{attribute 'linkalways'} 
{attribute 'no_explicit_call' := 'This FB is a CLASS and must be accessed using methods or properties'}
{attribute 'enable_dynamic_creation'}
FUNCTION_BLOCK _USINT EXTENDS NumericDatatypeBase
VAR
	localData : USINT;
	activeData : REFERENCE TO USINT REF= localData;
END_VAR

PROPERTY PUBLIC Address : PVOID
GET
Address := ADR(activeData);
END_GET
END_PROPERTY

METHOD PUBLIC ClearReference
VAR_INPUT
END_VAR
activeData REF= localData;
END_METHOD

METHOD PUBLIC Clone : I_Datatype
VAR
    pClone : POINTER TO _USINT;
END_VAR
pClone := __NEW(_USINT(InitialValue := Value));
Clone := pClone^;
END_METHOD

METHOD FB_init : BOOL
VAR_INPUT
	bInitRetains : BOOL; // if TRUE, the retain variables are initialized (warm start / cold start)
	bInCopyCode : BOOL;  // if TRUE, the instance afterwards gets moved into the copy code (online change)
	InitialValue : USINT;
END_VAR
localData := InitialValue;
END_METHOD

PROPERTY PUBLIC IsEven : BOOL
GET
IsEven := (Value mod 2) = 0;
END_GET
END_PROPERTY

PROPERTY PUBLIC IsFloat : BOOL
GET
IsFloat := FALSE;
END_GET
END_PROPERTY

PROPERTY PUBLIC IsSigned : BOOL
GET
IsSigned := FALSE;
END_GET
END_PROPERTY

METHOD PUBLIC MakeReferenceTo
VAR_INPUT
	ReferenceTarget : REFERENCE TO USINT;
END_VAR
activeData REF= ReferenceTarget;
END_METHOD

PROPERTY PUBLIC MaxValue : USINT
GET
MaxValue :=  DatatypeLimits.USINT_MAX_VALUE;
END_GET
END_PROPERTY

PROPERTY PUBLIC MinValue : USINT
GET
MinValue := DatatypeLimits.USINT_MIN_VALUE;
END_GET
END_PROPERTY

METHOD PROTECTED SerializeMaxValue
VAR_INPUT
	Serializer : I_Serializer;
END_VAR
Serializer.AddUsint(MaxValue);
END_METHOD

METHOD PROTECTED SerializeMinValue
VAR_INPUT
	Serializer : I_Serializer;
END_VAR
Serializer.AddUsint(MinValue);
END_METHOD

METHOD PUBLIC SerializeWith
VAR_INPUT
	Serializer : I_Serializer;
END_VAR
Serializer.AddUsint(activeData);
END_METHOD

PROPERTY PUBLIC Size : UDINT
GET
Size := SIZEOF(activeData);
END_GET
END_PROPERTY

METHOD TryDeserializeFrom : BOOL
VAR_INPUT
	Deserializer : I_Deserializer;
	Feedback : I_DeserializerFeedback;
END_VAR
TryDeserializeFrom := Deserializer.TryGetUsint(activeData, Feedback);
END_METHOD

METHOD TryMakeReferenceTo : BOOL
VAR_INPUT
	Target : I_Datatype;
END_VAR
VAR
	pTargetData : POINTER TO USINT;
END_VAR
IF NOT (Target.TypeName = TypeName) THEN
	RETURN;
END_IF

pTargetData := Target.Address;
activeData REF= pTargetData^;
TryMakeReferenceTo := TRUE;
END_METHOD

PROPERTY PUBLIC TypeName : T_MAXSTRING
GET
TypeName := 'USINT';
END_GET
END_PROPERTY

PROPERTY PUBLIC Value : REFERENCE TO USINT
GET
Value REF= activeData;
END_GET
END_PROPERTY

END_FUNCTION_BLOCK

(* stored: Version 1.1.0.1, ProductVersion 3.1.4024.13
   POU _USINT: Id {81b2d143-2840-482b-be90-2ad76730b020}, SpecialFunc None
   Folder Constructor: Id {19646add-caa7-40a7-beba-6091cc8cc00a}
   Folder Protected: Id {cb0754f0-619e-420b-b97e-fcb613a6589b}
   Property Address: Id {464a3ec8-54e3-4560-a5eb-be48f5986008}
   Get Get: Id {60ea4a0a-80a4-48b7-b29c-d9918bfb874c}
   Method ClearReference: Id {782734e1-c07f-4a07-a6d2-816695d17aaf}
   Method Clone: Id {6ce2ad4a-fd45-4082-a661-2591e8cbfd65}
   Method FB_init: Id {cc80f8ba-70e9-45ef-9610-5e6965f9f535}
   Property IsEven: Id {b2201ee4-c48b-059f-004c-0a0e1915d545}
   Get Get: Id {289460ea-e6a3-0bbb-1a43-9ff24fd135e3}
   Property IsFloat: Id {80c0da12-0ca7-4195-bdd6-c4cf867c086a}
   Get Get: Id {ff429fa0-6fb6-4f38-b113-8862c78e0d14}
   Property IsSigned: Id {cebffb7f-099e-4c38-9df0-d81790598eb5}
   Get Get: Id {0f041d57-d487-49ac-919b-0aee1f716557}
   Method MakeReferenceTo: Id {65699936-c612-4391-b1c7-e01a7f62e9c4}
   Property MaxValue: Id {c7d9343a-12f0-46fd-a438-5b9ead747e3e}
   Get Get: Id {7662962b-096d-4ba1-9dbb-4ae17c93d5c1}
   Property MinValue: Id {70a48e60-18a4-46c1-b5f7-d5135c0b64fe}
   Get Get: Id {7b9c61b7-92e3-46d4-8c2c-f898f837db6f}
   Method SerializeMaxValue: Id {3fa17023-84c4-4e10-b794-ed2d41025171}
   Method SerializeMinValue: Id {d59157fa-3028-4da0-843d-fb8f027861ea}
   Method SerializeWith: Id {71237bb9-2232-4637-b97a-0ffae93c88c9}
   Property Size: Id {ea2a4846-4552-47d4-9619-a96719e19fcc}
   Get Get: Id {37d4852b-045f-4ede-9ba0-7d16c6b3ef3e}
   Method TryDeserializeFrom: Id {2f28e960-7175-4644-a33a-6456d37fed4f}
   Method TryMakeReferenceTo: Id {6f2fb658-f821-4ac5-b639-be66a298a345}
   Property TypeName: Id {0484dc82-8fca-4dec-b049-648062144459}
   Get Get: Id {30ccebb5-7e44-4a4d-a905-6b09d7473636}
   Property Value: Id {85963213-01e6-4a65-b2d2-0663c27fb817}
   Get Get: Id {1ee2e363-1235-47a9-aec0-fa0314471208} *)
